// TIA Portal V16 export
// export: Created 2023-03-29T11:03:43.1290328Z, ExportSetting WithDefaults, DisplayName Totally Integrated Automation Portal, DisplayVersion V16 Update 6, DisplayName TIA Portal Version Control Interface, DisplayVersion V16 Update 2, DisplayName TIA Portal Openness, DisplayVersion V16 Update 6, DisplayName STEP 7 Professional, DisplayVersion V16 Update 6, DisplayName STEP 7 Safety, DisplayVersion V16, DisplayName WinCC Advanced, DisplayVersion V16 Update 6
DATA_BLOCK "Parametryzacja"   // DB12
TITLE = Konfiguracja parametrów
{ S7_Optimized_Access := 'FALSE' }
AUTHOR : rtecmer
VERSION : 0.1
// Dane konfiguracji parametrów przepływomierza, sond pomiarowych, przetworników
// stored: AutoNumber true, DBAccessibleFromOPCUA true, IsOnlyStoredInLoadMemory false, IsWriteProtectedInAS false
   VAR RETAIN
      "Setting analog" : Struct   // Parametry przetworników analogowych
         maxPrzepływomierz_Q2 : Real := 600.0;   // nastawa konfiguracji przetwornika przepływomierza wartość max przepływ
         minPrzepływomierz_Q2 : Real := 0.0;   // nastawa konfiguracji przetwornika przepływomierza wartość min przepływ
         maxPrzetwornikCiśnienia_B5 : Real := 16.0;   // nastawa konfiguracji przetwornika
         minPrzetwornikCiśnienia_B5 : Real := 0.0;   // nastawa konfiguracji przetwornika
         maxSondaHydro : Real := 1000.0;   // nastawa konfiguracji przetwornika
         minSondaHydro : Real := 0.0;   // nastawa konfiguracji przetwornika
      END_STRUCT;
      "Setting Controll" : Struct   // Parametry nastaw w procesie sterowania
         alarmMin_CiśnienieGranica : Real := 6.5;   // minimalne dopuszczalne ciśnienie Granica
         alarmMax_CiśnienieGranica : Real := 10.0;   // minimalne dopuszczalne ciśnienie Granica
         maxZbiorniki : Real := 600.0;   // stan alarmowy poziomu
         minZbiorniki : Real := 100.0;   // stan alarmowy poziomu
         max_położenie_Z10 : Real := 101.0;   // stan alarmowy położenia
         min_położenie_Z10 : Real := -0.5;   // stan alarmowy położenia
         setPoziomNapełniania : Real := 550.0;   // zadana wartość napełniania
         setPoziomOpróżnianai : Real := 30.0;   // zadana wartość opróżniania
         setPołożenieZ10 : Word;   // zadany [%] otwarcia
         tmpPołożenieZ10 : Word;   // tymczasowa zadany [%] otwarcia do przekazania
         ModelSterowania : Word;   // Zmienna przyjmująca wartość dziesiętnią oznaczającą model sterowania
         TrybSterowania : Word;   // Tryb 0-wyłączony, 1- Dobowy, 2- Tygodniowy, 3-Ręczny
      END_STRUCT;
      "Status drivers" : Struct   // Status napedów
         instZ1 : Word;   // status zasuwy
         instZ2 : Word;   // status zasuwy
         instZ3 : Word;   // status zasuwy
         instZ4 : Word;   // status zasuwy
         instZ5 : Word;   // status zasuwy
         instZ6 : Word;   // status zasuwy
         instZ7 : Word;   // status zasuwy
         instZ8 : Word;   // status zasuwy
         instZ9 : Word;   // status zasuwy
         instZ10 : Word;   // status zasuwy
      END_STRUCT;
      "Controls Tanks" : Struct   // Sterowanie zbiornikami
         aktywny_Zbiornik_1 : Bool;   // zbiornik włączony w cykl pracy 1=aktywny
         aktywny_Zbiornik_2 : Bool;   // zbiornik włączony w cykl pracy 1=aktywny
         aktywny_Zbiornik_3 : Bool;   // zbiornik włączony w cykl pracy 1=aktywny
         aktywny_Zbiornik_4 : Bool;   // zbiornik włączony w cykl pracy 1=aktywny
         aktywne_Napełnianie : Bool;   // bit aktywacji funkcji napełniania
         "aktywne _Przetłaczanie" : Bool;   // bit aktywacji funkcji przetłaczania
         aktywne_Dosilanie : Bool;   // bit aktywacji funkcji dosilania
      END_STRUCT;
      "Time Tanks" : Struct
         Start_napełnianie : DTL := DTL#1970-01-01-23:55:00;
         Stop_napełnianie : DTL := DTL#1970-01-01-16:00:00;
         Start_przetłaczanie_1 : DTL := DTL#1970-01-01-18:00:00;
         Stop_przetłaczanie_1 : DTL := DTL#1970-01-01-23:40:00;
         Start_dosilanie_1 : DTL := DTL#1970-01-01-18:00:00;
         Stop_dosilanie_1 : DTL := DTL#1970-01-01-23:40:00;
         Tank_bocking : Struct   // bity blokowania zbiornika w trybie sekwencyjnym
            blocing_tank1 : Bool;
            blocing_tank2 : Bool := false;
            blocing_tank3 : Bool := false;
            blocing_tank4 : Bool := false;
         END_STRUCT;
      END_STRUCT;
   END_VAR
BEGIN
END_DATA_BLOCK
